(* PLC project Unnamed, Unknown Unnamed 1 *)
(* stored: creationDateTime 2024-02-06T17:37:22, modificationDateTime 2024-02-11T17:53:41 *)

PROGRAM lab2
  VAR
    count AT %MW8 : INT;
    color0 AT %MW0 : INT;
    color1 AT %MW1 : INT;
    color2 AT %MW2 : INT;
    color3 AT %MW3 : INT;
    color4 AT %MW4 : INT;
    color5 AT %MW5 : INT;
    color6 AT %MW6 : INT;
    color7 AT %MW7 : INT;
    red_anode AT %QX100.0 : BOOL;
    green_anode AT %QX100.1 : BOOL;
    blue_anode AT %QX100.2 : BOOL;
    button AT %IX100.0 : BOOL;
    mode AT %QX0.0 : BOOL;
  END_VAR
  VAR
    TON0 : TON;
    TON1 : TON;
    count_en : BOOL;
    auto_count_en : BOOL;
    CTU0 : CTU;
    CTU_Res : BOOL;
    Mux_Out : INT;
  END_VAR
  VAR  (* added by the conversion: wires and edge detectors of the diagram *)
    R_TRIG1 : R_TRIG;
  END_VAR

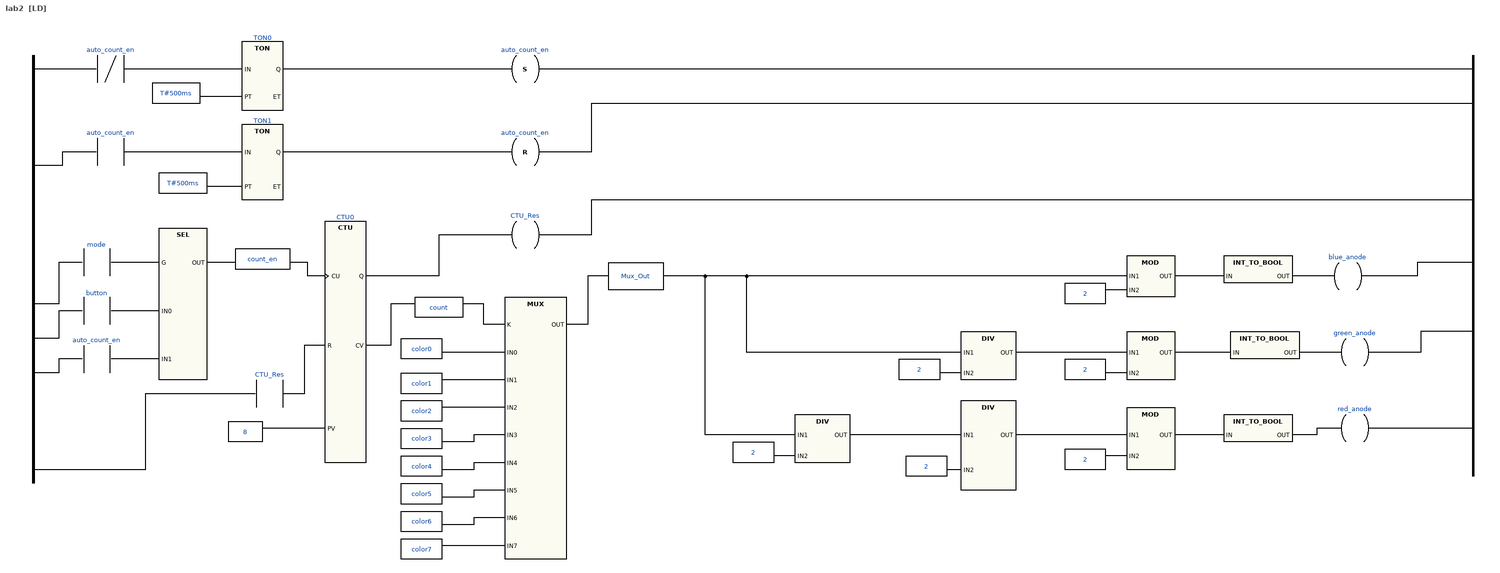
(* LD diagram, written out as Structured Text *)
TON0(IN := NOT auto_count_en, PT := T#500ms);
IF TON0.Q THEN auto_count_en := TRUE; END_IF;
TON1(IN := auto_count_en, PT := T#500ms);
IF TON1.Q THEN auto_count_en := FALSE; END_IF;
R_TRIG1(CLK := count_en);
CTU0(CU := R_TRIG1.Q, R := CTU_Res, PV := 8);
CTU_Res := CTU0.Q;
count_en := SEL(mode, button, auto_count_en);
Mux_Out := MUX(count, color0, color1, color2, color3, color4, color5, color6, color7);
blue_anode := INT_TO_BOOL(Mux_Out MOD 2);
count := CTU0.CV;
green_anode := INT_TO_BOOL(Mux_Out / 2 MOD 2);
red_anode := INT_TO_BOOL(Mux_Out / 2 / 2 MOD 2);
END_PROGRAM

CONFIGURATION Config0
  RESOURCE Res0 ON PLC
    TASK task0(INTERVAL := T#20ms, PRIORITY := 0);
    PROGRAM instance0 WITH task0 : lab2;
  END_RESOURCE
END_CONFIGURATION
